FUNCTION_BLOCK Process EXTENDS Station IMPLEMENTS IProcess
VAR_INPUT
END_VAR
VAR_OUTPUT
END_VAR
VAR
	_isProcess : BOOL;
	_startPos : MC_LREAL;
	_endPos : MC_LREAL;
	_processVelo : MC_LREAL;
END_VAR

PROPERTY EndPosition : MC_LREAL
GET
EndPosition := _endPos;
END_GET
SET
_endPos := EndPosition;
END_SET
END_PROPERTY

{warning 'add property implementation'}
PROPERTY IsProcess : BOOL
GET
IsProcess := _isProcess;
END_GET
SET
_isProcess := IsProcess;
END_SET
END_PROPERTY

PROPERTY ProcessVelocity : MC_LREAL
GET
ProcessVelocity := _processVelo;
END_GET
SET
_processVelo := ProcessVelocity;
END_SET
END_PROPERTY

PROPERTY StartPosition : MC_LREAL
GET
StartPosition := _startPos;
END_GET
SET
_startPos := StartPosition;
END_SET
END_PROPERTY

END_FUNCTION_BLOCK

(* stored: Version 1.1.0.1, ProductVersion 3.1.4024.11
   POU Process: Id {d2e75364-5fbc-4562-a2ad-425968d5f182}, SpecialFunc None
   Property EndPosition: Id {65043570-5e02-48d8-bfb0-5c560a6a952b}
   Get Get: Id {bf2122ca-6425-4989-ac27-0984d8a65701}
   Set Set: Id {0e8c8642-fded-4757-a3b6-3759eea005c6}
   Property IsProcess: Id {82549bd7-942d-4761-8c09-dc22c9d610d0}
   Get Get: Id {180f94a2-c956-4574-91d5-be594d5ef0a4}
   Set Set: Id {9b7659f1-97bf-4aa7-8dbb-ec0417c43521}
   Property ProcessVelocity: Id {8eba20b0-3bc9-4dc7-a15d-1c2c3523cee6}
   Get Get: Id {3c55315f-6a68-4740-9e8d-06477ef7e1c9}
   Set Set: Id {de5929c4-8559-470c-8c9f-203a033d0a7d}
   Property StartPosition: Id {bd94f458-cdf0-4d8f-8006-f91599da287b}
   Get Get: Id {f2433651-b5e9-4e44-bcc7-c17df437db39}
   Set Set: Id {a8c55751-3793-42e7-bc09-430e0d686ffc} *)
